Fanuc KAREL source: kt00071.KL

PROGRAM KT00071
%NOLOCKGROUP
VAR
I1:INTEGER
H2 : ARRAY[2] OF SHORT
OUT:INTEGER
BEGIN
I1=2
H2[1]=3
OUT=(I1*H2[1])
END KT00071
